(* Logix 5000 project; controller ABB_Drive_Test vendor 1 type 14 code 149 rev 33.12; software revision 33.01; part 4 of 6 *)
(* tags used below, declared in another part *)
   append : BOOL;
   bytestring : STRING;
   CF_del : TIMER;
   cmdto : BOOL;
   extra_info : BOOL;
   f_nr : DINT;
   falctrl01 : CONTROL;
   flush_delay : TIMER;
   intsource : INT[100];
   MSGtriggers : DINT;
   next_file_response : FS_response;
   prev_index : DINT;
   searchstring : STRING;
   spacestring : STRING;
   step : DINT;
   tempDINT : DINT;
   tempDINTAR : DINT[10];
   CF0x3MSG : MESSAGE;   // detect card
   CF0x4fMSG : MESSAGE;   // read from file
   CF0x50MSG : MESSAGE;   // write to file
   CF0x52MSG : MESSAGE;   // file open
   CF0x53MSG : MESSAGE;   // set file pointer
   CF0x54MSG : MESSAGE;   // file close
   CF0x55MSG : MESSAGE;   // delete file
   CF0x56MSG : MESSAGE;   // create directory
   CF0x57MSG : MESSAGE;   // rename/move file
   CF0x58MSG : MESSAGE;   // Find first file
   CF0x59MSG : MESSAGE;   // Find next file
   CF0x5aMSG : MESSAGE;   // Find close
   CF_data : SINT[512];
   CF_RW_functions : CF_functions;
(* CF_FunctionsProgram, continued *)

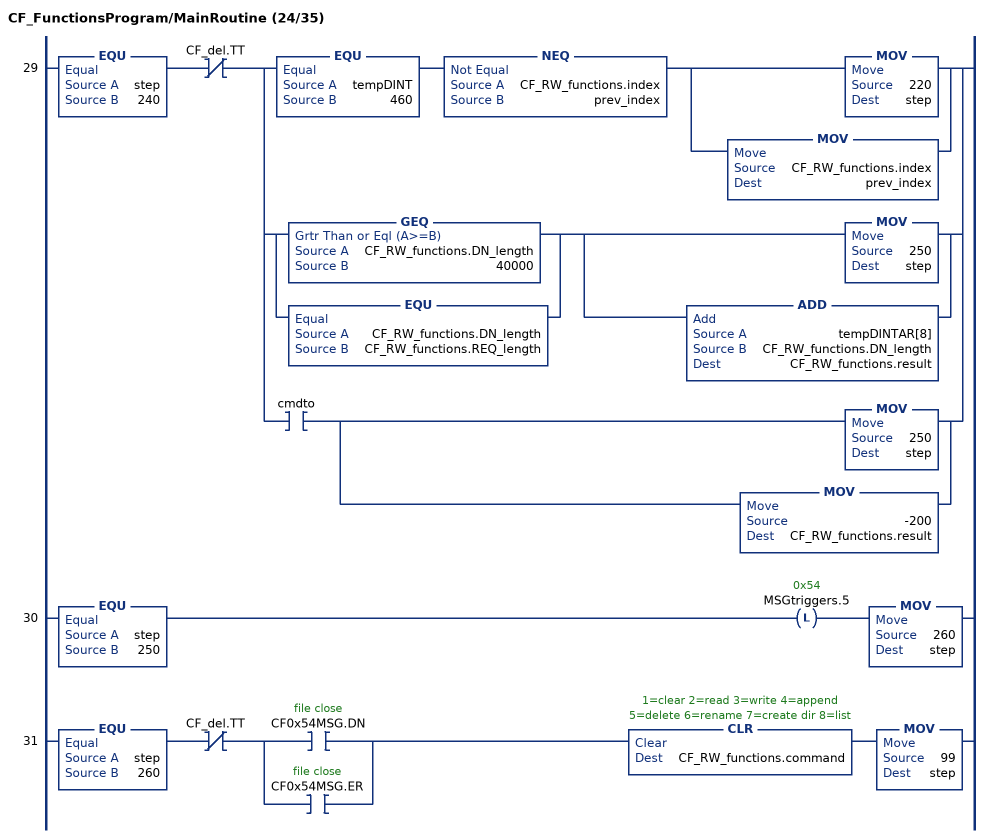
   29: EQU(step,240)XIO(CF_del.TT)[EQU(tempDINT,460) NEQ(CF_RW_functions.index,prev_index) [MOV(220,step) ,MOV(CF_RW_functions.index,prev_index) ] ,[GEQ(CF_RW_functions.DN_length,40000) ,EQU(CF_RW_functions.DN_length,CF_RW_functions.REQ_length) ] [MOV(250,step) ,ADD(tempDINTAR[8],CF_RW_functions.DN_length,CF_RW_functions.result) ] ,XIC(cmdto) [MOV(250,step) ,MOV(-200,CF_RW_functions.result) ] ];
   30: EQU(step,250)OTL(MSGtriggers.5)MOV(260,step);
   31: EQU(step,260)XIO(CF_del.TT)[XIC(CF0x54MSG.DN) ,XIC(CF0x54MSG.ER) ]CLR(CF_RW_functions.command)MOV(99,step);
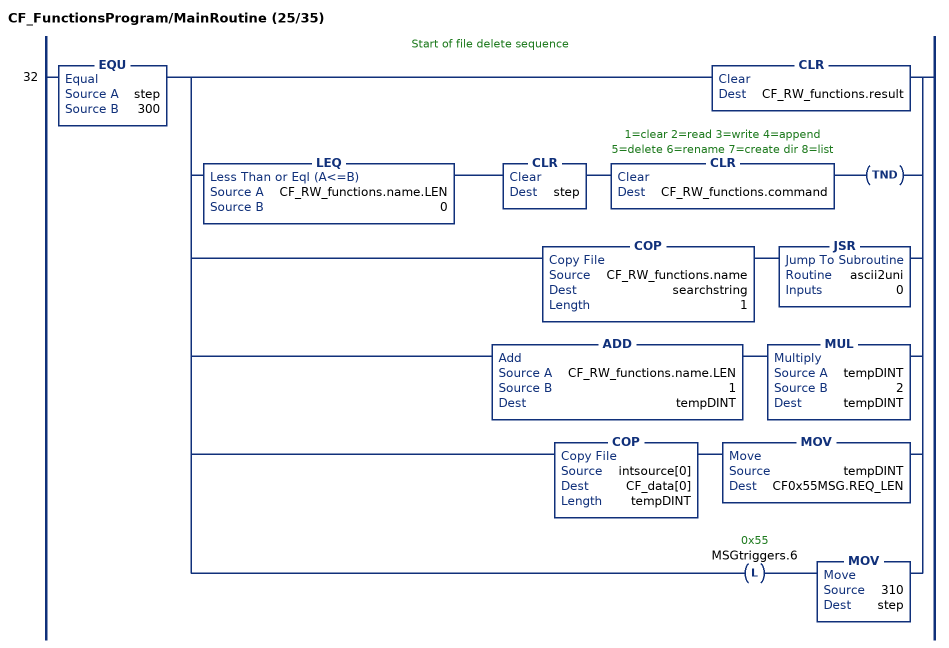
   // Start of file delete sequence
   32: EQU(step,300)[CLR(CF_RW_functions.result) ,LEQ(CF_RW_functions.name.LEN,0) CLR(step) CLR(CF_RW_functions.command) TND() ,COP(CF_RW_functions.name,searchstring,1) JSR(ascii2uni,0) ,ADD(CF_RW_functions.name.LEN,1,tempDINT) MUL(tempDINT,2,tempDINT) ,COP(intsource[0],CF_data[0],tempDINT) MOV(tempDINT,CF0x55MSG.REQ_LEN) ,OTL(MSGtriggers.6) MOV(310,step) ];
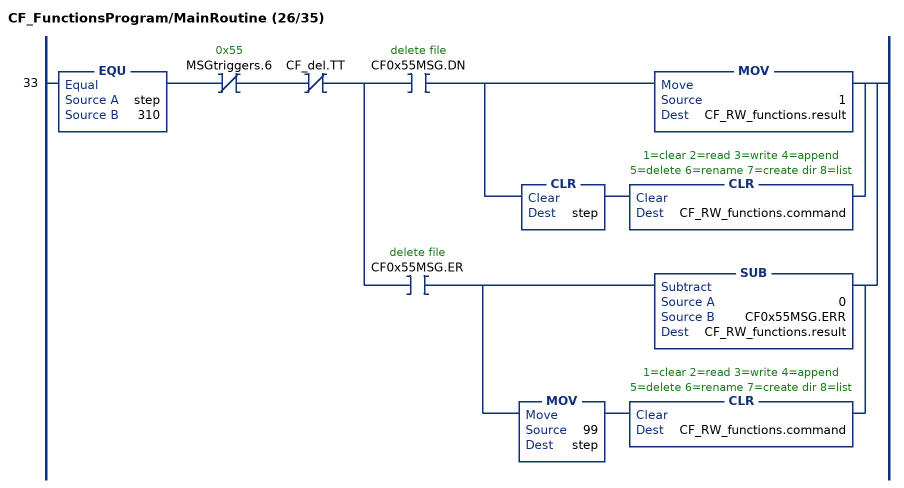
   33: EQU(step,310)XIO(MSGtriggers.6)XIO(CF_del.TT)[XIC(CF0x55MSG.DN) [MOV(1,CF_RW_functions.result) ,CLR(step) CLR(CF_RW_functions.command) ] ,XIC(CF0x55MSG.ER) [SUB(0,CF0x55MSG.ERR,CF_RW_functions.result) ,MOV(99,step) CLR(CF_RW_functions.command) ] ];
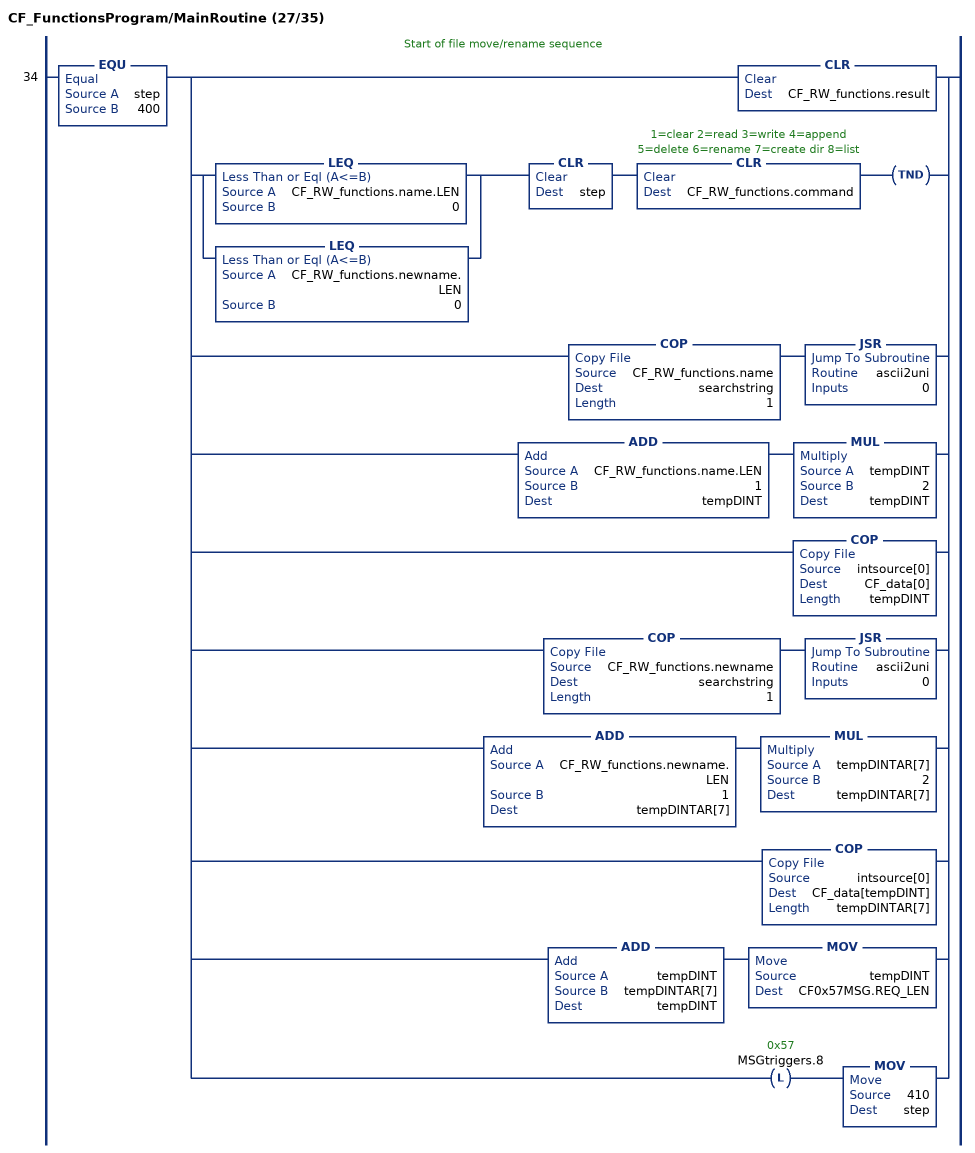
   // Start of file move/rename sequence
   34: EQU(step,400)[CLR(CF_RW_functions.result) ,[LEQ(CF_RW_functions.name.LEN,0) ,LEQ(CF_RW_functions.newname.LEN,0) ] CLR(step) CLR(CF_RW_functions.command) TND() ,COP(CF_RW_functions.name,searchstring,1) JSR(ascii2uni,0) ,ADD(CF_RW_functions.name.LEN,1,tempDINT) MUL(tempDINT,2,tempDINT) ,COP(intsource[0],CF_data[0],tempDINT) ,COP(CF_RW_functions.newname,searchstring,1) JSR(ascii2uni,0) ,ADD(CF_RW_functions.newname.LEN,1,tempDINTAR[7]) MUL(tempDINTAR[7],2,tempDINTAR[7]) ,COP(intsource[0],CF_data[tempDINT],tempDINTAR[7]) ,ADD(tempDINT,tempDINTAR[7],tempDINT) MOV(tempDINT,CF0x57MSG.REQ_LEN) ,OTL(MSGtriggers.8) MOV(410,step) ];
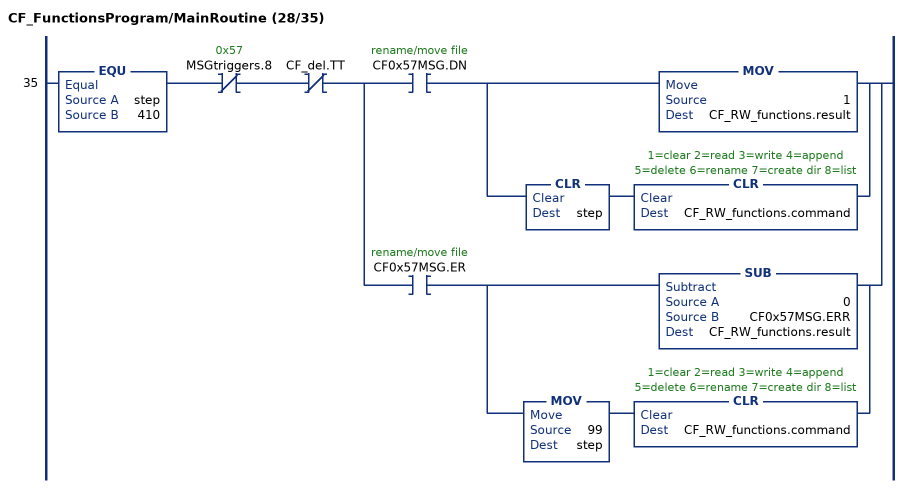
   35: EQU(step,410)XIO(MSGtriggers.8)XIO(CF_del.TT)[XIC(CF0x57MSG.DN) [MOV(1,CF_RW_functions.result) ,CLR(step) CLR(CF_RW_functions.command) ] ,XIC(CF0x57MSG.ER) [SUB(0,CF0x57MSG.ERR,CF_RW_functions.result) ,MOV(99,step) CLR(CF_RW_functions.command) ] ];
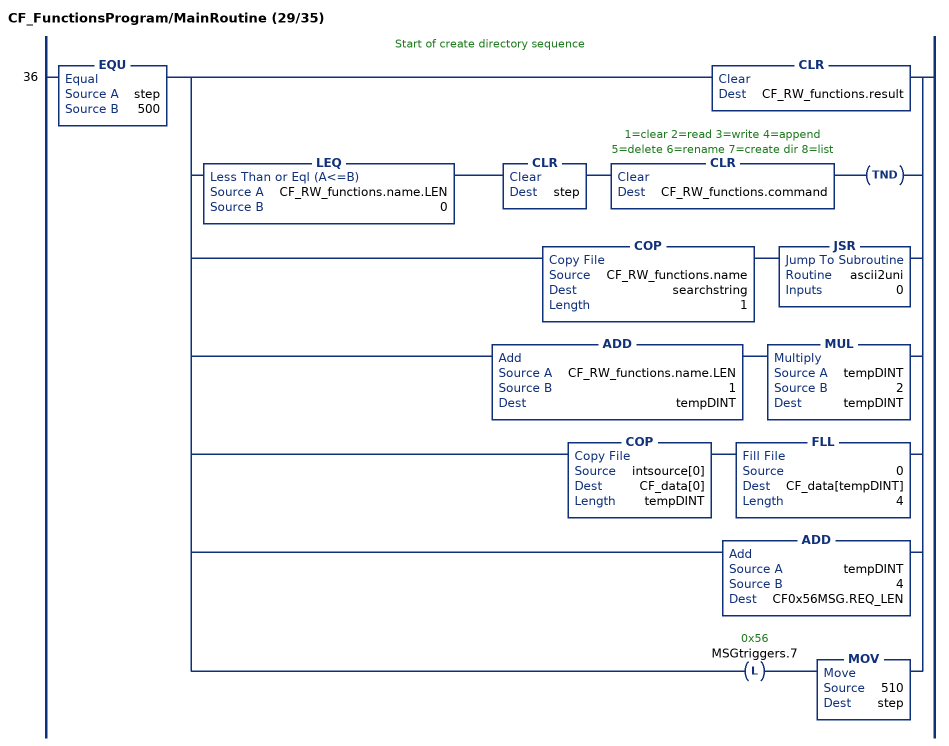
   // Start of create directory sequence
   36: EQU(step,500)[CLR(CF_RW_functions.result) ,LEQ(CF_RW_functions.name.LEN,0) CLR(step) CLR(CF_RW_functions.command) TND() ,COP(CF_RW_functions.name,searchstring,1) JSR(ascii2uni,0) ,ADD(CF_RW_functions.name.LEN,1,tempDINT) MUL(tempDINT,2,tempDINT) ,COP(intsource[0],CF_data[0],tempDINT) FLL(0,CF_data[tempDINT],4) ,ADD(tempDINT,4,CF0x56MSG.REQ_LEN) ,OTL(MSGtriggers.7) MOV(510,step) ];
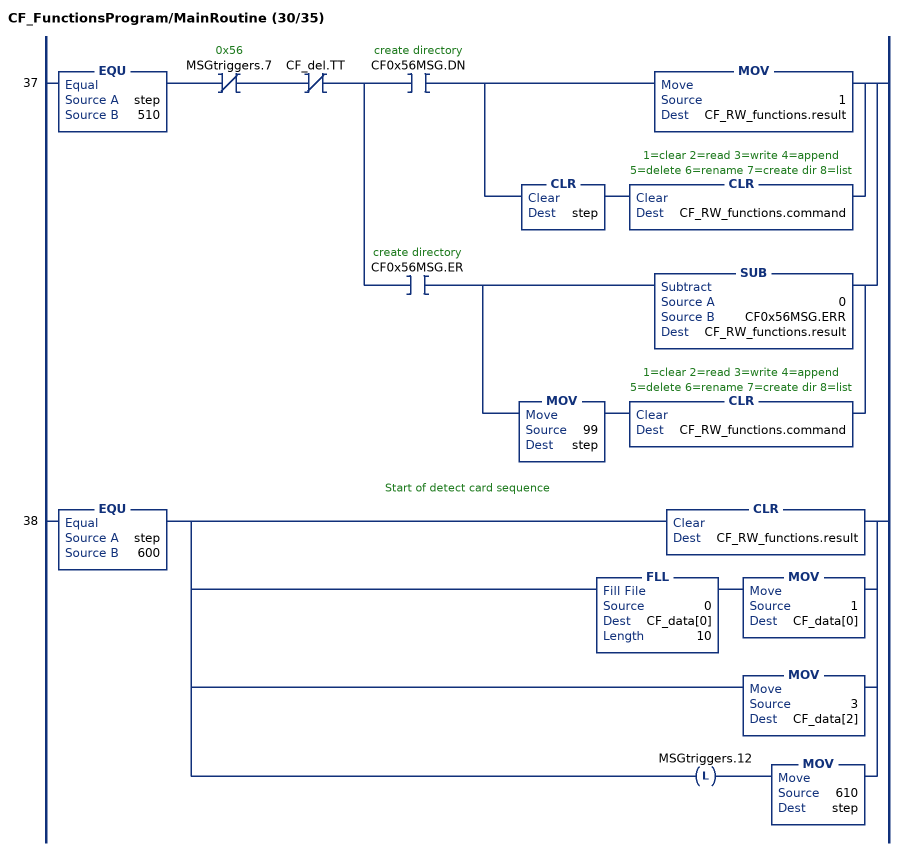
   37: EQU(step,510)XIO(MSGtriggers.7)XIO(CF_del.TT)[XIC(CF0x56MSG.DN) [MOV(1,CF_RW_functions.result) ,CLR(step) CLR(CF_RW_functions.command) ] ,XIC(CF0x56MSG.ER) [SUB(0,CF0x56MSG.ERR,CF_RW_functions.result) ,MOV(99,step) CLR(CF_RW_functions.command) ] ];
   // Start of detect card sequence
   38: EQU(step,600)[CLR(CF_RW_functions.result) ,FLL(0,CF_data[0],10) MOV(1,CF_data[0]) ,MOV(3,CF_data[2]) ,OTL(MSGtriggers.12) MOV(610,step) ];
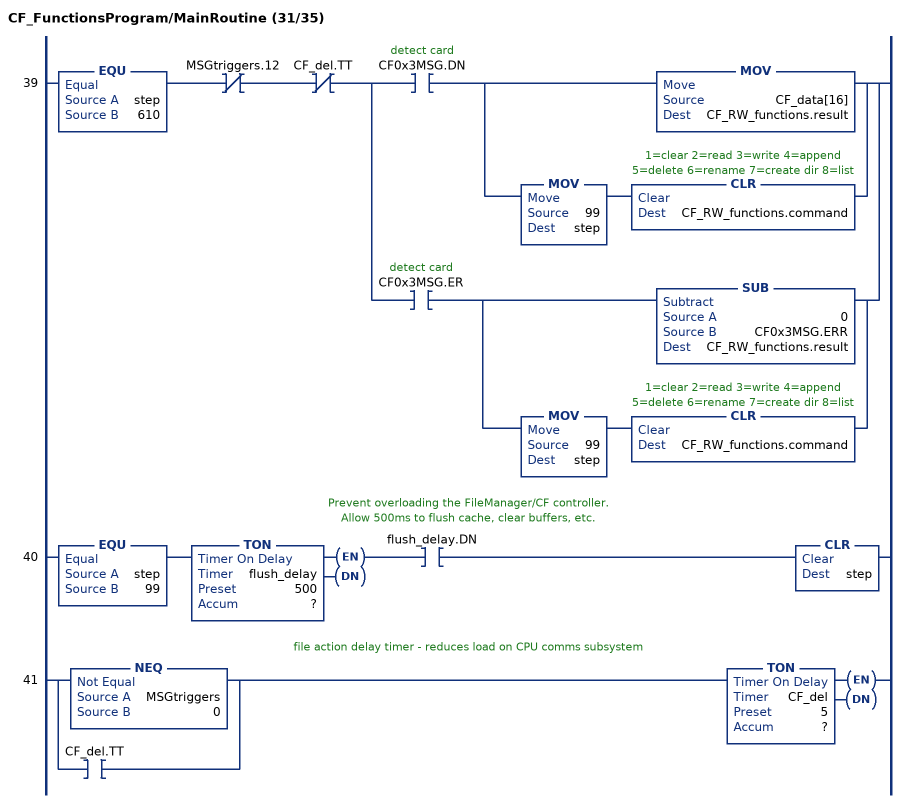
   39: EQU(step,610)XIO(MSGtriggers.12)XIO(CF_del.TT)[XIC(CF0x3MSG.DN) [MOV(CF_data[16],CF_RW_functions.result) ,MOV(99,step) CLR(CF_RW_functions.command) ] ,XIC(CF0x3MSG.ER) [SUB(0,CF0x3MSG.ERR,CF_RW_functions.result) ,MOV(99,step) CLR(CF_RW_functions.command) ] ];
   // Prevent overloading the FileManager/CF controller.
   // Allow 500ms to flush cache, clear buffers, etc.
   40: EQU(step,99)TON(flush_delay,?,?)XIC(flush_delay.DN)CLR(step);
   // file action delay timer - reduces load on CPU comms subsystem
   41: [NEQ(MSGtriggers,0) ,XIC(CF_del.TT) ]TON(CF_del,?,?);
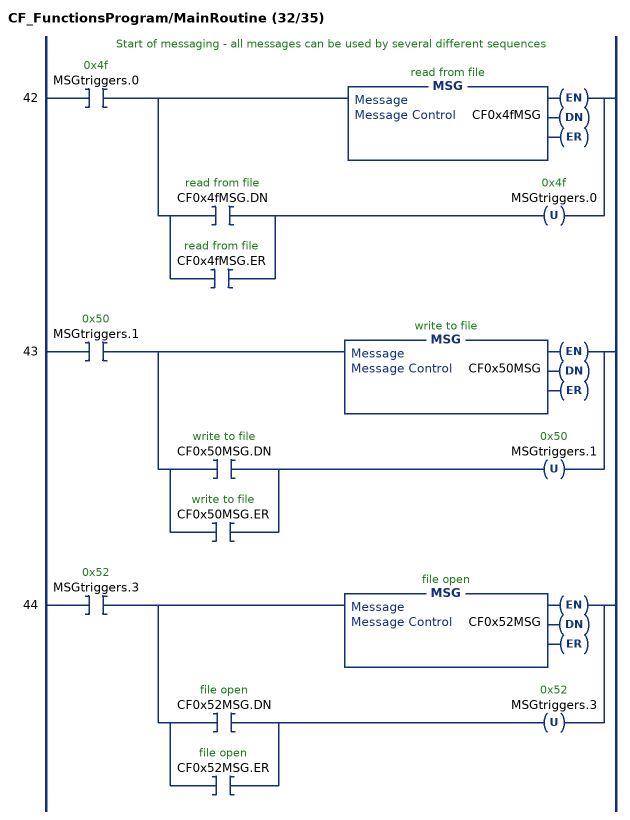
   // Start of messaging - all messages can be used by several different sequences
   42: XIC(MSGtriggers.0)[MSG(CF0x4fMSG) ,[XIC(CF0x4fMSG.DN) ,XIC(CF0x4fMSG.ER) ] OTU(MSGtriggers.0) ];
   43: XIC(MSGtriggers.1)[MSG(CF0x50MSG) ,[XIC(CF0x50MSG.DN) ,XIC(CF0x50MSG.ER) ] OTU(MSGtriggers.1) ];
   44: XIC(MSGtriggers.3)[MSG(CF0x52MSG) ,[XIC(CF0x52MSG.DN) ,XIC(CF0x52MSG.ER) ] OTU(MSGtriggers.3) ];
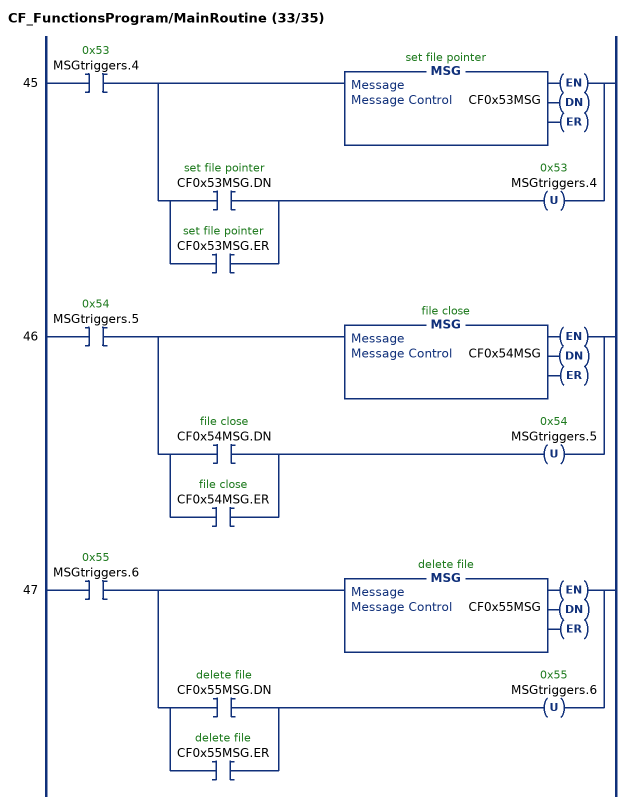
   45: XIC(MSGtriggers.4)[MSG(CF0x53MSG) ,[XIC(CF0x53MSG.DN) ,XIC(CF0x53MSG.ER) ] OTU(MSGtriggers.4) ];
   46: XIC(MSGtriggers.5)[MSG(CF0x54MSG) ,[XIC(CF0x54MSG.DN) ,XIC(CF0x54MSG.ER) ] OTU(MSGtriggers.5) ];
   47: XIC(MSGtriggers.6)[MSG(CF0x55MSG) ,[XIC(CF0x55MSG.DN) ,XIC(CF0x55MSG.ER) ] OTU(MSGtriggers.6) ];
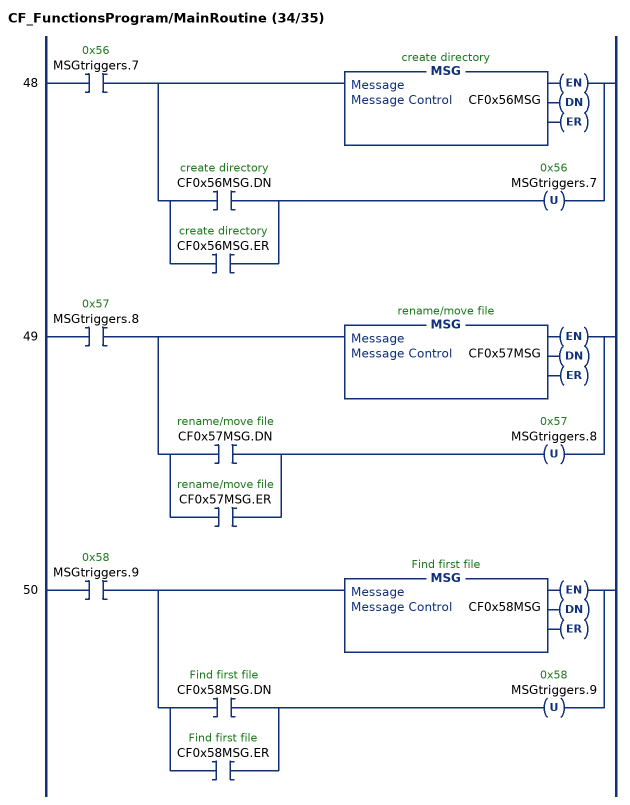
   48: XIC(MSGtriggers.7)[MSG(CF0x56MSG) ,[XIC(CF0x56MSG.DN) ,XIC(CF0x56MSG.ER) ] OTU(MSGtriggers.7) ];
   49: XIC(MSGtriggers.8)[MSG(CF0x57MSG) ,[XIC(CF0x57MSG.DN) ,XIC(CF0x57MSG.ER) ] OTU(MSGtriggers.8) ];
   50: XIC(MSGtriggers.9)[MSG(CF0x58MSG) ,[XIC(CF0x58MSG.DN) ,XIC(CF0x58MSG.ER) ] OTU(MSGtriggers.9) ];
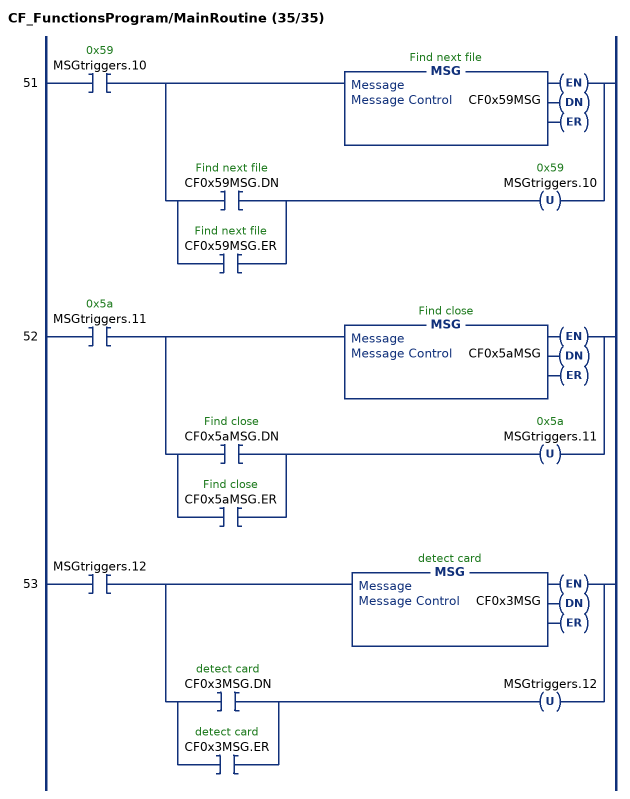
   51: XIC(MSGtriggers.10)[MSG(CF0x59MSG) ,[XIC(CF0x59MSG.DN) ,XIC(CF0x59MSG.ER) ] OTU(MSGtriggers.10) ];
   52: XIC(MSGtriggers.11)[MSG(CF0x5aMSG) ,[XIC(CF0x5aMSG.DN) ,XIC(CF0x5aMSG.ER) ] OTU(MSGtriggers.11) ];
   53: XIC(MSGtriggers.12)[MSG(CF0x3MSG) ,[XIC(CF0x3MSG.DN) ,XIC(CF0x3MSG.ER) ] OTU(MSGtriggers.12) ];
END_ROUTINE

ROUTINE unic2ascii   (* ladder *)
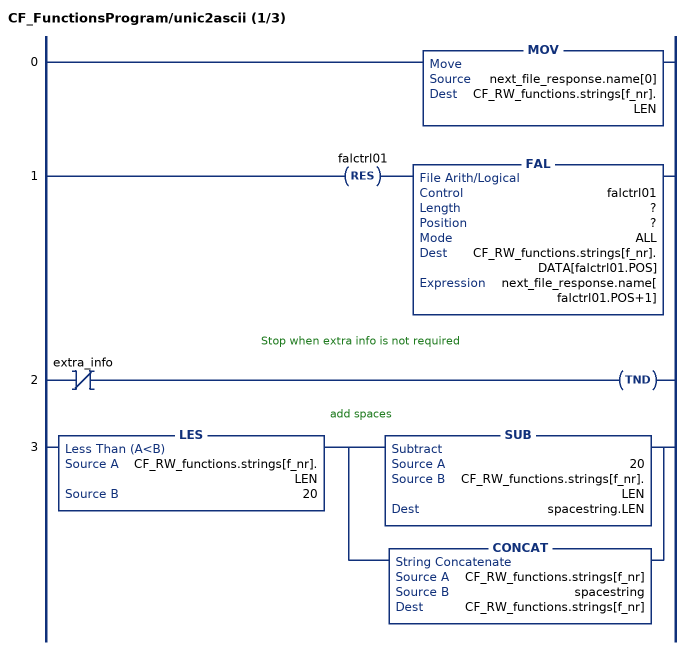
   0: MOV(next_file_response.name[0],CF_RW_functions.strings[f_nr].LEN);
   1: RES(falctrl01)FAL(falctrl01,?,?,ALL,CF_RW_functions.strings[f_nr].DATA[falctrl01.POS],next_file_response.name[falctrl01.POS+1]);
   // Stop when extra info is not required
   2: XIO(extra_info)TND();
   // add spaces
   3: LES(CF_RW_functions.strings[f_nr].LEN,20)[SUB(20,CF_RW_functions.strings[f_nr].LEN,spacestring.LEN) ,CONCAT(CF_RW_functions.strings[f_nr],spacestring,CF_RW_functions.strings[f_nr]) ];
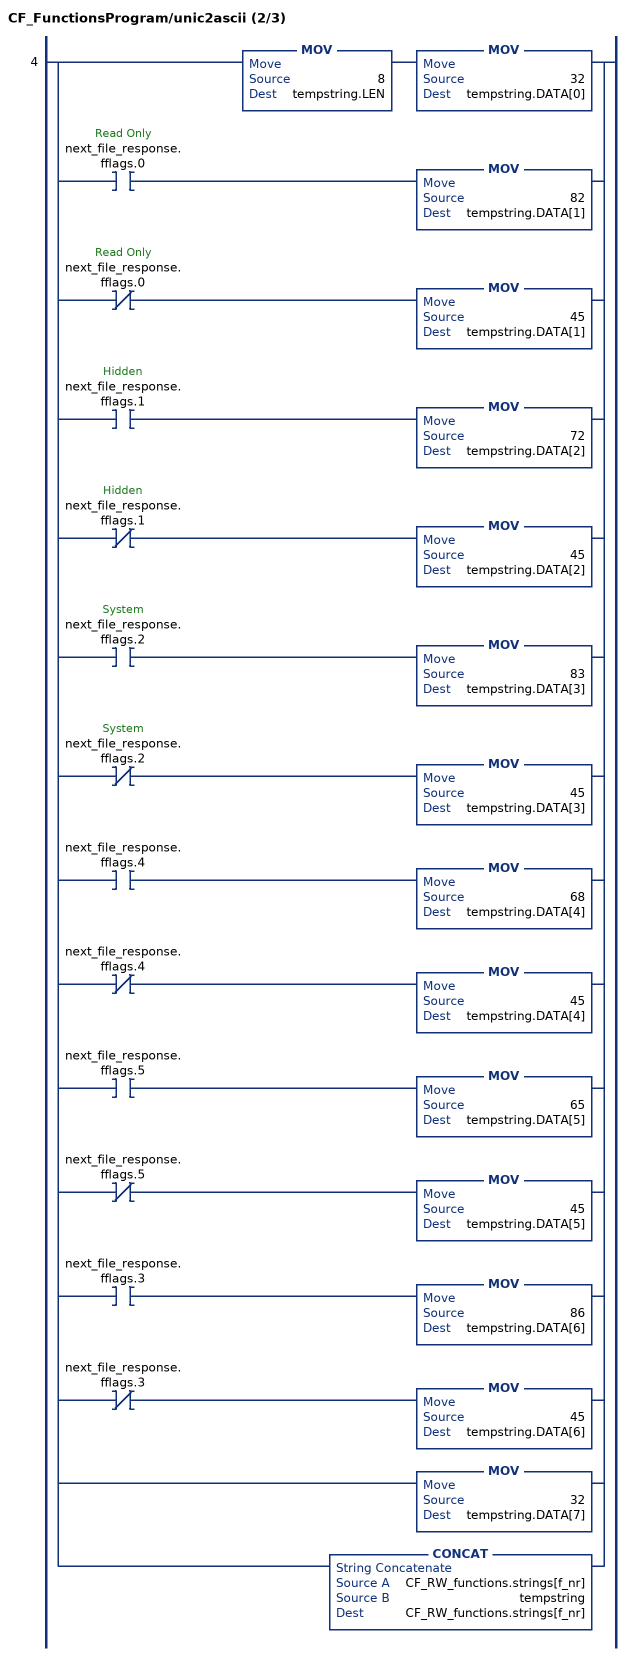
   4: [MOV(8,tempstring.LEN) MOV(32,tempstring.DATA[0]) ,XIC(next_file_response.fflags.0) MOV(82,tempstring.DATA[1]) ,XIO(next_file_response.fflags.0) MOV(45,tempstring.DATA[1]) ,XIC(next_file_response.fflags.1) MOV(72,tempstring.DATA[2]) ,XIO(next_file_response.fflags.1) MOV(45,tempstring.DATA[2]) ,XIC(next_file_response.fflags.2) MOV(83,tempstring.DATA[3]) ,XIO(next_file_response.fflags.2) MOV(45,tempstring.DATA[3]) ,XIC(next_file_response.fflags.4) MOV(68,tempstring.DATA[4]) ,XIO(next_file_response.fflags.4) MOV(45,tempstring.DATA[4]) ,XIC(next_file_response.fflags.5) MOV(65,tempstring.DATA[5]) ,XIO(next_file_response.fflags.5) MOV(45,tempstring.DATA[5]) ,XIC(next_file_response.fflags.3) MOV(86,tempstring.DATA[6]) ,XIO(next_file_response.fflags.3) MOV(45,tempstring.DATA[6]) ,MOV(32,tempstring.DATA[7]) ,CONCAT(CF_RW_functions.strings[f_nr],tempstring,CF_RW_functions.strings[f_nr]) ];
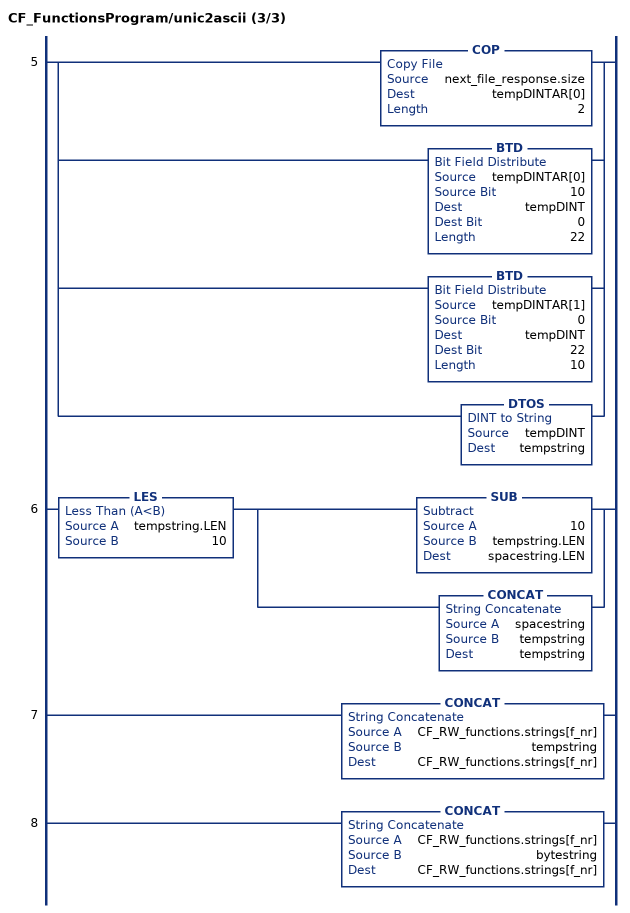
   5: [COP(next_file_response.size,tempDINTAR[0],2) ,BTD(tempDINTAR[0],10,tempDINT,0,22) ,BTD(tempDINTAR[1],0,tempDINT,22,10) ,DTOS(tempDINT,tempstring) ];
   6: LES(tempstring.LEN,10)[SUB(10,tempstring.LEN,spacestring.LEN) ,CONCAT(spacestring,tempstring,tempstring) ];
   7: CONCAT(CF_RW_functions.strings[f_nr],tempstring,CF_RW_functions.strings[f_nr]);
   8: CONCAT(CF_RW_functions.strings[f_nr],bytestring,CF_RW_functions.strings[f_nr]);
END_ROUTINE
END_PROGRAM

PROGRAM CSVProgram   (* main routine MainRoutine *)
VAR
   ad_pointer : DINT := 256;
   cf_bigWcmd01 : DINT;
   cf_bigWoffset01 : DINT := 5120;
   cfbw01 : CF_big_write := (array_offset := 5120);
   check_log_age : BOOL;
   d1hf_copy : BOOL;
   DataIndex : DINT := 10;
   dayms : DINT := 35452354;
   dayms_frac : REAL := 0.09363253;
   daysince1900 : DINT := 35888;
   daysinprevmonths : DINT[13] := ([0] := 366, [2] := 31, [3] := 59, [4] := 90, [5] := 121, [6] := 151, [7] := 181, [8] := 212, [9] := 243, [10] := 273, [11] := 304, [12] := 334);
   detect_1st_half_full : BOOL;
   filename : STRING := 'Log_1998_04_03_02_11.csv';
   filename_end : STRING := '.csv';
   filenamestart : STRING := 'Log_';
   get_filesize : BOOL;
   ldt : DateTime := (year := 1998, month := 4, day := 3, hour := 2, minute := 14, second := 49, usec := 850360);
   log_check_active : BOOL;
   logfile_size : DINT := 25216;
   logging_enabled : BOOL := 1;   // HABILITAR DATALOGGER
   logpulse : BOOL;
   max_file_size : DINT := 250000;
   max_logfiles : DINT := 75;
   nr_of_logfiles : DINT := 75;
   nr_of_writes : DINT := 9;
   ofdindex : DINT;
   ofdoldestfilename : STRING;
   ofdoldestTS : DINT := 999999999;
   ofdSEQ : DINT;
   sec_pulse : TIMER := (PRE := 987654321, ACC := 909, EN := 1, TT := 1);
   tempstring : STRING := '1.00000000$0D$0A';
   testfilename : BOOL;
   tmpDINT : DINT := 2;
   trigger_write : BOOL;
   write_1st_half : BOOL;
   write_length : DINT := 4992;
   write_offset : DINT := 5120;
   wrSEQ : DINT;
   Year_1901 : DINT := 97;
END_VAR

ROUTINE DeleteOldestLogFile   (* ladder *)
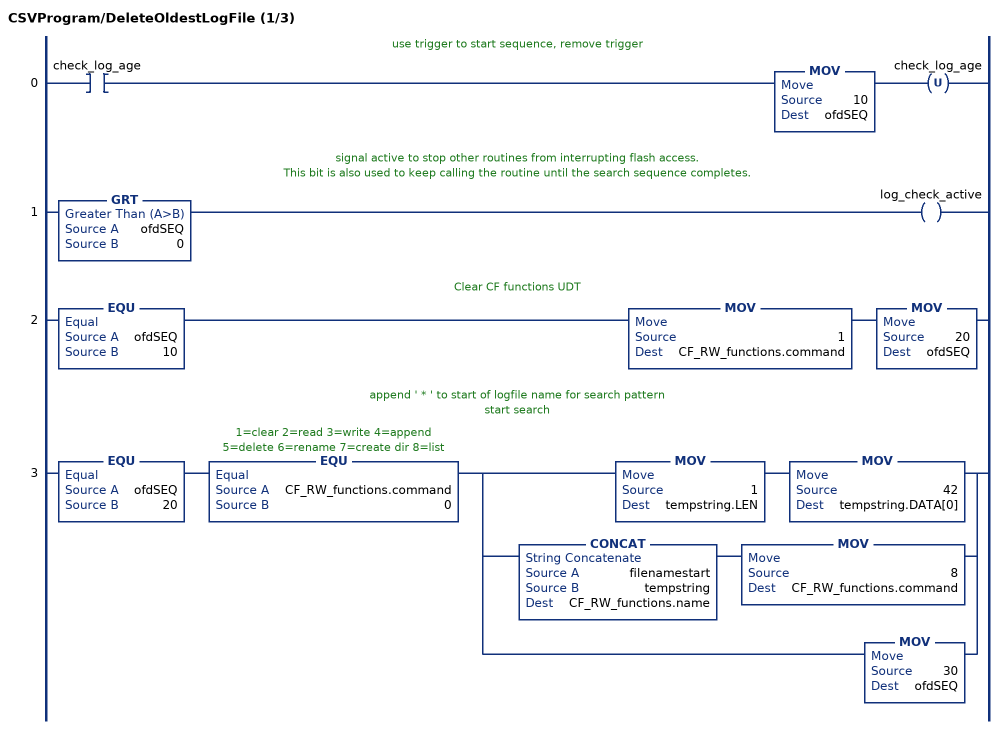
   // use trigger to start sequence, remove trigger
   0: XIC(check_log_age)MOV(10,ofdSEQ)OTU(check_log_age);
   // signal active to stop other routines from interrupting flash access.
   // This bit is also used to keep calling the routine until the search sequence completes.
   1: GRT(ofdSEQ,0)OTE(log_check_active);
   // Clear CF functions UDT
   2: EQU(ofdSEQ,10)MOV(1,CF_RW_functions.command)MOV(20,ofdSEQ);
   // append ' * ' to start of logfile name for search pattern
   // start search
   3: EQU(ofdSEQ,20)EQU(CF_RW_functions.command,0)[MOV(1,tempstring.LEN) MOV(42,tempstring.DATA[0]) ,CONCAT(filenamestart,tempstring,CF_RW_functions.name) MOV(8,CF_RW_functions.command) ,MOV(30,ofdSEQ) ];
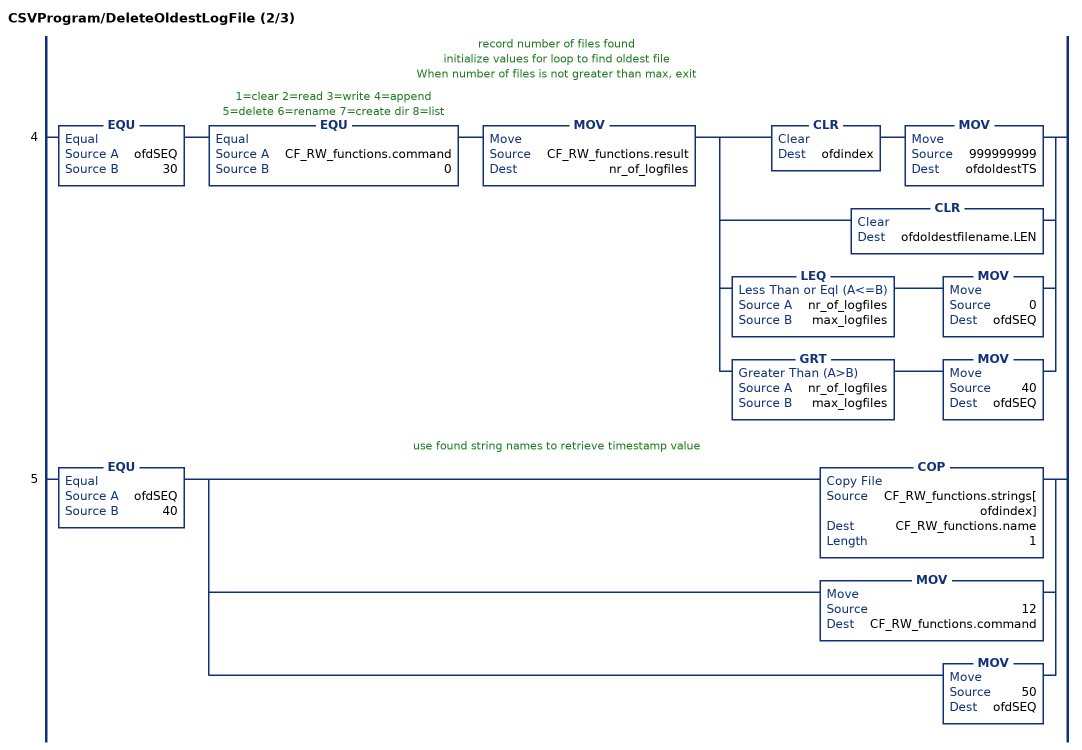
   // record number of files found
   // initialize values for loop to find oldest file
   // When number of files is not greater than max, exit
   4: EQU(ofdSEQ,30)EQU(CF_RW_functions.command,0)MOV(CF_RW_functions.result,nr_of_logfiles)[CLR(ofdindex) MOV(999999999,ofdoldestTS) ,CLR(ofdoldestfilename.LEN) ,LEQ(nr_of_logfiles,max_logfiles) MOV(0,ofdSEQ) ,GRT(nr_of_logfiles,max_logfiles) MOV(40,ofdSEQ) ];
   // use found string names to retrieve timestamp value
   5: EQU(ofdSEQ,40)[COP(CF_RW_functions.strings[ofdindex],CF_RW_functions.name,1) ,MOV(12,CF_RW_functions.command) ,MOV(50,ofdSEQ) ];
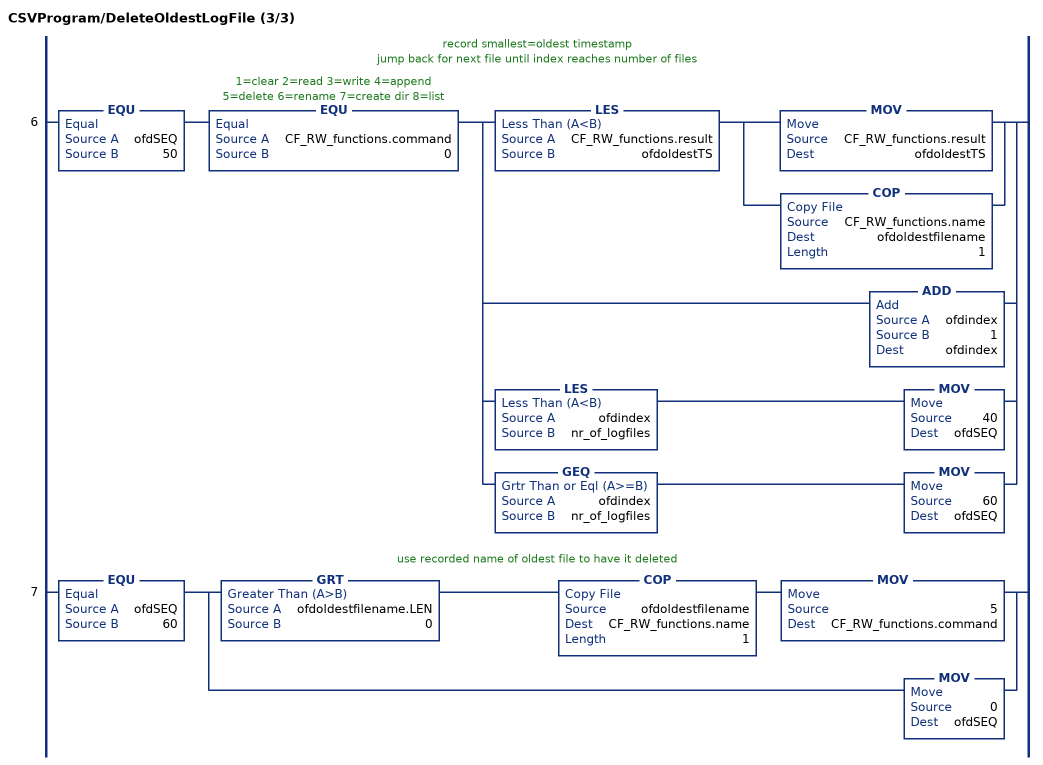
   // record smallest=oldest timestamp
   // jump back for next file until index reaches number of files
   6: EQU(ofdSEQ,50)EQU(CF_RW_functions.command,0)[LES(CF_RW_functions.result,ofdoldestTS) [MOV(CF_RW_functions.result,ofdoldestTS) ,COP(CF_RW_functions.name,ofdoldestfilename,1) ] ,ADD(ofdindex,1,ofdindex) ,LES(ofdindex,nr_of_logfiles) MOV(40,ofdSEQ) ,GEQ(ofdindex,nr_of_logfiles) MOV(60,ofdSEQ) ];
   // use recorded name of oldest file to have it deleted
   7: EQU(ofdSEQ,60)[GRT(ofdoldestfilename.LEN,0) COP(ofdoldestfilename,CF_RW_functions.name,1) MOV(5,CF_RW_functions.command) ,MOV(0,ofdSEQ) ];
END_ROUTINE
